PROGRAM Main
VAR
    (*
    // Test Pitch Control
    fbPitchControl : FB_PitchControl;
    TestPitch : HOMS_PitchMechanism := (ReqPosLimHi:=2000,
                                        ReqPosLimLo:=-2000,
                                        diEncPosLimHi:=10768330,
                                        diEncPosLimLo:=8141680);
    M1 : ST_MotionStage;
    bPitchDone : BOOL;
    *)

    // Test Bender vs No Bender
    TESTWithBender : DUT_HOMS;
    M1 : ST_MotionStage := (nEnableMode:=ENUM_StageEnableMode.ALWAYS);
    M2 : ST_MotionStage := (nEnableMode:=ENUM_StageEnableMode.ALWAYS);
    M3 : ST_MotionStage := (nEnableMode:=ENUM_StageEnableMode.ALWAYS);
    M4 : ST_MotionStage := (nEnableMode:=ENUM_StageEnableMode.ALWAYS);
    M5 : ST_MotionStage := (nEnableMode:=ENUM_StageEnableMode.ALWAYS);
    M6 : ST_MotionStage := (nEnableMode:=ENUM_StageEnableMode.ALWAYS);
    fbBender : FB_Bender;

    fbMotionStage_m1 : FB_MotionStage;
    fbMotionStage_m2 : FB_MotionStage;
    fbMotionStage_m3 : FB_MotionStage;
    fbMotionStage_m4 : FB_MotionStage;
    fbMotionStage_m6 : FB_MotionStage;
END_VAR

(*
// Test Pitch Control
M1.bLimitBackwardEnable;
M1.bLimitForwardEnable;
M1.bHardwareEnable;
M1.fVelocity := 150.0;
fbPitchControl(Pitch:=TestPitch,
               Stepper:=M1,
               lrCurrentSetpoint:=M1.fPosition,
               q_bDone=>bPitchDone,
               q_bBusy=>);
IF NOT M1.bHardwareEnable THEN
    M1.fPosition := M1.stAxisStatus.fActPosition;
END_IF
*)

// Test Bender vs. No Bender:
// M1L0
M1.bLimitForwardEnable := TRUE;
M1.bLimitBackwardEnable := TRUE;
M1.bPowerSelf := TRUE;

M2.bLimitForwardEnable := TRUE;
M2.bLimitBackwardEnable := TRUE;
M2.bPowerSelf := TRUE;

M3.bLimitForwardEnable := TRUE;
M3.bLimitBackwardEnable := TRUE;
M3.bPowerSelf := TRUE;

M4.bLimitForwardEnable := TRUE;
M4.bLimitBackwardEnable := TRUE;
M4.bPowerSelf := TRUE;

M5.bLimitForwardEnable := TRUE;
M5.bLimitBackwardEnable := TRUE;
M5.bPowerSelf := TRUE;

M6.bLimitForwardEnable := TRUE;
M6.bLimitBackwardEnable := TRUE;
M6.bPowerSelf := TRUE;
TESTWithBender.fbRunHOMS(stYup:=M1,
                         stYdwn:=M2,
                         stXup:=M3,
                         stXdwn:=M4,
                         stPitch:=M5,
                         nYupEncRef:=0,
                         nYdwnEncRef:=0,
                         nXupEncRef:=0,
                         nXdwnEncRef:=0,
                         bExecuteCoupleY:=TESTWithBender.bExecuteCoupleY,
                         bExecuteCoupleX:=TESTWithBender.bExecuteCoupleX,
                         bExecuteDecoupleY:=TESTWithBender.bExecuteDecoupleY,
                         bExecuteDecoupleX:=TESTWithBender.bExecuteDecoupleX,
                         bGantryAlreadyCoupledY=>TESTWithBender.bGantryAlreadyCoupledY,
                         bGantryAlreadyCoupledX=>TESTWithBender.bGantryAlreadyCoupledX,
                         nCurrGantryY=>TESTWithBender.nCurrGantryY,
                         nCurrGantryX=>TESTWithBender.nCurrGantryX);
fbBender(stBender:=M6,
         bSTOEnable1:=TESTWithBender.fbRunHOMS.bSTOEnable1,
         bSTOEnable2:=TESTWithBender.fbRunHOMS.bSTOEnable2);

fbMotionStage_m1(stMotionStage:=M1);
fbMotionStage_m2(stMotionStage:=M2);
fbMotionStage_m3(stMotionStage:=M3);
fbMotionStage_m4(stMotionStage:=M4);
fbMotionStage_m6(stMotionStage:=M6);

END_PROGRAM

(* stored: Version 1.1.0.1, ProductVersion 3.1.4024.12
   POU Main: Id {bced800e-adc0-4347-8ec8-808d3a0afec0}, SpecialFunc None *)
